// TwinCAT 3 PLC project Development
// ProgramVersion: 3.1.4026.14
// CompilerDefines: release,VISU_USEPROPERTYINFO
// libraries:
//   Tc2_Drive, * (Beckhoff Automation GmbH)
//   Tc2_EtherCAT, * (Beckhoff Automation GmbH)
//   Tc2_MC2, * (Beckhoff Automation GmbH)
//   Tc2_MC2_Drive, * (Beckhoff Automation GmbH)
//   Tc2_Standard, * (Beckhoff Automation GmbH)
//   Tc2_System, * (Beckhoff Automation GmbH)
//   Tc2_Utilities, * (Beckhoff Automation GmbH)
//   Tc3_Element, * (Zerlauth)
//   Tc3_IPCDiag, * (Beckhoff Automation GmbH)
//   Tc3_Module, * (Beckhoff Automation GmbH)
// project tree:
//   GVLs/ IO.TcGVL (not stored)
//   InDevelopment/Axis/ FB_Axis.TcPOU (not stored), F_TcError.TcPOU (not stored), I_Axis.TcIO (not stored)
//   InDevelopment/Contactor/ FB_Contactor.TcPOU
//   InDevelopment/Cylinder/ FB_Cylinder.TcPOU, ST_CylinderOptions.TcDUT (not stored)
//   InDevelopment/ FB_ComponentEX.TcPOU, FB_EthercatDiagnostic.TcPOU (not stored)
//   InDevelopment/PnozMulti/ FB_PnozMulti.TcPOU
//   Modules/ FB_Module01.TcPOU, FB_Machine.TcPOU (not stored), FB_Module02.TcPOU
//   / PlcTask.TcTTO (not stored)
//   POUs/ FB_ComponentT.TcPOU, MAIN.TcPOU
// real-time tasks:
//   TASK PlcTask: cycle T#500ms, priority 21, ADS port 351
//   TASK UnitTestTask: cycle T#1ms, priority 1, ADS port 350
// motion (NC):
//   TASK NC-Task 1 SAF: cycle T#2ms, priority 4, ADS port 501
//   TASK NC-Task 1 SVB: cycle T#10ms, priority 8, ADS port 511
//   AXIS Achse 1 (id 1)
//     OtherSettings: AllowMotionCmdToSlave=true
//     encoder EncType=1
//     drive DrvType=5
//       Analog: TorqueSetpointScale=10, ScaleFactorActTorque=0.1
//       TimeComp: TaskDelayCycles=1
//     controller CtrType=1
//       CtrPara: PriorControlFactor=1
//         Observer: BandWidth=20
// I/O:
//   DEVICE Gerät 1 (EtherCAT) (disabled), AmsNetId 10.58.50.38.2.1
//     Klemme 1 (EK1100) [EK1100 EtherCAT-Koppler (2A E-Bus)]
//     Box 2 (EP1008-0001) [EP1008-0001 8 K. Dig. Eingang 24V, 3ms, M8]
// variable links:
//   Development/Development Instance <-> Device 1 (EtherCAT)
//     PlcTask Inputs/MAIN.fbMachine.fbEthercatDiagnostic.AmsNetID <-> InfoData/AmsNetId

// ---- InDevelopment/Contactor/FB_Contactor.TcPOU
FUNCTION_BLOCK FB_Contactor EXTENDS FB_Element
VAR_INPUT
	bInput				AT%I*: BOOL;
END_VAR
VAR_OUTPUT
	bOutput				AT%I*: BOOL;
END_VAR
VAR
END_VAR

super^();

METHOD PROTECTED M_Running
IF bOutput THEN
	IF bInput  THEN
		;
	ELSE
		P_Event.M_Fatal('Feedback wrong state %s', 0);		
	END_IF
END_IF
END_METHOD

METHOD PROTECTED M_Starting : BOOL (* Return state complete*)
IF bOutput THEN
	IF bInput THEN
		M_Starting:= TRUE;
	ELSE
		P_Event.M_Fatal('Feedback wrong state %s', 0);
	END_IF
ELSE
	IF bInput THEN
		P_Event.M_Fatal('Feedback wrong state %s', 0);
	ELSE
		bOutput:= TRUE;
	END_IF	
	
END_IF
END_METHOD

END_FUNCTION_BLOCK

// ---- InDevelopment/Cylinder/FB_Cylinder.TcPOU
FUNCTION_BLOCK FB_Cylinder EXTENDS FB_Element
VAR_INPUT
	stOptions:				ST_CylinderOptions;
END_VAR
VAR_OUTPUT
END_VAR
VAR
	bInHomePosition			AT%I*:		BOOL;
	bInWorkPosition			AT%I*:		BOOL;
	bToHomePosition			AT%Q*:		BOOL;
	bToWorkPosition			AT%Q*:		BOOL;
	fbHomePositon:			FB_Debounce;
	fbWorkPositon:			FB_Debounce;
	fbStarup:				TON;
	fbTimeout:				TON;
END_VAR

SUPER^();

METHOD PROTECTED M_Aborting : BOOL (* Return*)
bToHomePosition:= FALSE;
bToWorkPosition:= FALSE;
M_Aborting:= TRUE;
END_METHOD

METHOD PROTECTED M_Execute : BOOL // Return state complete
VAR_INPUT
END_VAR
fbHomePositon(bInput:= bInHomePosition);
fbWorkPositon(bInput:= bInWorkPosition);
fbTimeout(PT:= stOptions.tTimeout);
END_METHOD

METHOD PROTECTED M_Starting : BOOL // Return state complete
VAR_INPUT
END_VAR
IF SUPER^.M_Starting() THEN
	fbHomePositon.tTime:= stOptions.tDebounce;
	fbWorkPositon.tTime:= stOptions.tDebounce;
	// Check positons
	IF bToHomePosition AND bToWorkPosition THEN
		IF stOptions.tStartup <> T#0S THEN
			fbStarup(In:= TRUE, PT:= stOptions.tStartup);
			IF fbStarup.Q THEN
				fbStarup(In:= FALSE);
				bToHomePosition:= FALSE;
				bToWorkPosition:= FALSE;
				M_Starting:= TRUE;		
			END_IF
		ELSE
			M_Starting:= TRUE;	
		END_IF
	ELSIF bToHomePosition THEN
		IF NOT bInHomePosition THEN
			P_Event.M_AddSTRING(fbReflection.P_ID);
			P_Event.M_AddSTRING(stOptions.sHomePosition);
			P_Event.M_Error('Cylinder not in Home Positon (%s-%s)', 0);
		ELSIF bInWorkPosition THEN
			P_Event.M_AddSTRING(fbReflection.P_ID);
			P_Event.M_AddSTRING(stOptions.sWorkPosition);
			P_Event.M_Error('Cylinder in Work Positon (%s-%s)', 0);
		ELSE
			M_Starting:= TRUE;	
		END_IF
	ELSIF bToWorkPosition THEN
		IF NOT bInWorkPosition THEN
			P_Event.M_AddSTRING(fbReflection.P_ID);
			P_Event.M_AddSTRING(stOptions.sWorkPosition);
			P_Event.M_Error('Cylinder not in Work Positon (%s-%s)', 0);				
		ELSIF bInHomePosition THEN
			P_Event.M_AddSTRING(fbReflection.P_ID);
			P_Event.M_AddSTRING(stOptions.sHomePosition);
			P_Event.M_Error('Cylinder not in Home Positon (%s-%s)', 0);
		ELSE
			M_Starting:= TRUE;	
		END_IF
	ELSE
		IF bInWorkPosition THEN
			bToWorkPosition:= TRUE;
			M_Starting:= TRUE;
		ELSIF bInHomePosition THEN
			bToHomePosition:= TRUE;
			M_Starting:= TRUE;
		ELSIF stOptions.tStartup <> T#0S THEN		
			bToHomePosition:= TRUE;
			bToWorkPosition:= TRUE;
		ELSE
			M_Starting:= TRUE;
		END_IF
	END_IF
END_IF
END_METHOD

METHOD PUBLIC M_ToHome : BOOL
VAR_INPUT
END_VAR
IF bToWorkPosition THEN
	fbTimeout(IN:= FALSE);
	bToHomePosition:= TRUE;
	bToWorkPosition:= FALSE;

ELSIF bToHomePosition  THEN
	IF NOT fbWorkPositon.P_Value AND fbHomePositon.P_Value THEN
		M_ToHome:= TRUE;
	ELSE
		fbTimeout.IN:= TRUE;
		IF fbTimeout.Q THEN
			IF fbWorkPositon.P_Value THEN
				P_Event.M_AddSTRING(fbReflection.P_ID);
				P_Event.M_AddSTRING(stOptions.sWorkPosition);
				P_Event.M_Error('Cylinder Work Positon not left (%s%s)', 1120);				

			ELSIF NOT fbHomePositon.P_Value THEN
				P_Event.M_AddSTRING(fbReflection.P_ID);
				P_Event.M_AddSTRING(stOptions.sWorkPosition);
				P_Event.M_Error('Cylinder Home Positon not reached (%s%s)', 1121);
	
			END_IF
		END_IF
	END_IF
END_IF
END_METHOD

METHOD PUBLIC M_ToWork : BOOL
VAR_INPUT
END_VAR
IF bToHomePosition THEN
	fbTimeout(IN:= FALSE);
	bToHomePosition:= FALSE;
	bToWorkPosition:= TRUE;	

ELSIF bToWorkPosition  THEN
	IF fbWorkPositon.P_Value AND NOT fbHomePositon.P_Value THEN
		M_ToWork:= TRUE;
	ELSE
		fbTimeout.IN:= TRUE;
		IF fbTimeout.Q THEN
			IF NOT fbWorkPositon.P_Value THEN
				P_Event.M_AddSTRING(fbReflection.P_ID);
				P_Event.M_AddSTRING(stOptions.sWorkPosition);
				P_Event.M_Error('Cylinder Work Positon not reached (%s%s)', 1122);				

			ELSIF fbHomePositon.P_Value THEN
				P_Event.M_AddSTRING(fbReflection.P_ID);
				P_Event.M_AddSTRING(stOptions.sWorkPosition);
				P_Event.M_Error('Cylinder Home Positon not left (%s%s)', 1122);		

			END_IF
		END_IF
	END_IF
END_IF
END_METHOD

{attribute 'suppress_wrn_C0410'}
PROPERTY PUBLIC P_Options : REFERENCE TO ST_CylinderOptions
GET
P_Options ref= stOptions;
END_GET
END_PROPERTY

END_FUNCTION_BLOCK

// ---- InDevelopment/FB_ComponentEX.TcPOU
FUNCTION_BLOCK FB_ComponentEX EXTENDS FB_Element
VAR_INPUT
END_VAR
VAR_OUTPUT
END_VAR
VAR
	bError:			BOOL;
	bAbort:			BOOL;
	bStop:			BOOL;
	bInformation:	BOOL;
	bWarning:		BOOL;
END_VAR

SUPER^();

METHOD PROTECTED M_Execute : BOOL
VAR_INPUT
END_VAR
CASE fbSequence.P_Number OF
	E_Sequence.Start:
		fbSequence.M_Await('Start', 0, T#0S, T#0S, TRUE, TRUE, 10);
	
	10:
		fbSequence.M_Await('Step 10',0,  T#0S, T#0S, TRUE, TRUE, 20);
		
	20:
		fbSequence.M_Await('Step 20',0,  T#0S, T#0S, FALSE, TRUE, E_Sequence.Done);	
		
	E_Sequence.Done:
		fbSequence.M_Reset();
		
END_CASE

IF bAbort THEN
	bAbort:= FALSE;
	fbEvent.M_AddSTRING('1');
	fbEvent.M_AddSTRING('2');
	fbEvent.M_AddSTRING('3');
	fbEvent.M_Fatal('First Error Abort %s %s %s', 6);
END_IF

IF bStop THEN
	bStop:= FALSE;
	fbEvent.M_AddSTRING('a');
	fbEvent.M_AddSTRING('b');
	fbEvent.M_AddSTRING('c');
	fbEvent.M_Error('First Error Stop', 7);
END_IF

IF bInformation THEN
	fbEvent.M_Info('Info', 12);	
END_IF

IF bWarning THEN
	fbEvent.M_Warning('Warning', 13);	
END_IF
END_METHOD

END_FUNCTION_BLOCK

// ---- InDevelopment/PnozMulti/FB_PnozMulti.TcPOU
FUNCTION_BLOCK FB_PnozMulti EXTENDS FB_Element
VAR_INPUT
END_VAR
VAR_OUTPUT
END_VAR
VAR
	bOK:					BOOL:= TRUE;
	bReset:					BOOL;
	fbReset:				TON:= (PT:= T#1S);
END_VAR

SUPER^();

METHOD PROTECTED M_Resetting : BOOL // Return state complete
VAR_INPUT
END_VAR
SUPER^.M_Resetting();
bReset:= TRUE;
fbReset(IN:= TRUE, PT:= T#1S);
IF fbReset.Q THEN
	bReset:= FALSE;
	M_Resetting:= TRUE;
END_IF
END_METHOD

METHOD PROTECTED M_Running
IF NOT bOK THEN
	P_Event.M_AddSTRING(fbReflection.P_ID);
	P_Event.M_Fatal('PnozMulti no ok Signal (%s)', 0);
END_IF
END_METHOD

END_FUNCTION_BLOCK

// ---- Modules/FB_Module01.TcPOU
FUNCTION_BLOCK FB_Module01 EXTENDS FB_Module
VAR_INPUT
END_VAR
VAR_OUTPUT
END_VAR
VAR
END_VAR

// https://peterzerlauth.com/
SUPER^();

METHOD PROTECTED M_Running
VAR_INPUT
END_VAR
END_METHOD

METHOD PROTECTED M_Starting : BOOL
VAR_INPUT
END_VAR
M_Starting:= SUPER^.M_Starting();
END_METHOD

METHOD PROTECTED M_Stopping : BOOL // Return state complete
VAR_INPUT
END_VAR
// State Stopping
M_Stopping:= SUPER^.M_Stopping();
END_METHOD

END_FUNCTION_BLOCK

// ---- Modules/FB_Module02.TcPOU
FUNCTION_BLOCK FB_Module02 EXTENDS FB_Module
VAR_INPUT
END_VAR
VAR_OUTPUT
END_VAR
VAR
	fbPnozMulti:				FB_PnozMulti;
	fbComponent0:				FB_ComponentEx;
	fbComponent1:				FB_ComponentEx;
	fbContactor:				FB_Contactor;
	fbCylinder:					FB_Cylinder;
END_VAR

// https://peterzerlauth.com/
SUPER^();

fbComponent0();
fbComponent1();
fbContactor();
fbCylinder();
fbPnozMulti();

fbContactor.bInput:= fbContactor.bOutput;

METHOD PROTECTED M_Execute : BOOL
VAR_INPUT
END_VAR
VAR
	bReturn:					BOOL:= TRUE;
END_VAR
CASE fbSequence.P_Number OF
	E_Sequence.Start:
		bReturn:= TRUE;
		fbSequence.M_Await('Start 0', 0,  T#0S , T#1S, TRUE, bReturn, 10);
	
	10:
		bReturn:= TRUE;
		fbSequence.M_Await('Step 10', 0,  T#0S, T#0S, TRUE, bReturn, 20);
		
	20:
		bReturn:= TRUE;
		fbSequence.M_Await('Step 20', 0,  T#1S, T#0S, FALSE, bReturn, E_Sequence.Done);
		IF fbSequence.P_Timeout THEN
			fbEvent.M_Error('Overrride timeout error', 0);
		END_IF
		
	E_Sequence.Done:
		fbSequence.M_Reset();

END_CASE
END_METHOD

METHOD PROTECTED M_Idle : BOOL (* Return*)
SUPER^.M_Idle();

fbLevel4.M_Attach(fbPnozMulti);
fbLevel3.M_Attach(fbComponent0);
fbLevel3.M_Attach(fbComponent1);
fbLevel2.M_Attach(fbPnozMulti);
fbLevel2.M_Attach(fbContactor);
fbLevel1.M_Attach(fbCylinder);
END_METHOD

END_FUNCTION_BLOCK

// ---- POUs/FB_ComponentT.TcPOU
FUNCTION_BLOCK FB_ComponentT EXTENDS FB_Element
VAR_INPUT
END_VAR
VAR_OUTPUT
END_VAR
VAR
	bAbort: BOOL;
END_VAR

super^();

METHOD PROTECTED M_Execute : BOOL (* Return*)

IF bAbort THEN
	P_Event.M_Fatal('msg', 0);
END_IF
END_METHOD

END_FUNCTION_BLOCK

// ---- POUs/MAIN.TcPOU
PROGRAM MAIN
VAR
	bTest:				BOOL;
	fbMachine:			FB_Machine;
	fbModule1:			FB_Module01;
	fbModule2:			FB_Module02;
	
	fbComponent1:		FB_ComponentT;
	fbComponent2:		FB_ComponentT;	
	bInit: 				BOOL:= TRUE;
	exceptionCode: 		__SYSTEM.ExceptionCode;
	exception: 			__SYSTEM.ExceptionCode;
	fbFileLogger:		FB_FileLogger<10>:= (sPathName:= 'C:\Temp\log.txt');
	stEvent: 			Tc3_Element.ST_Event;
	bLog: BOOL;
END_VAR

bTest:= NOT bTest;

__TRY
	fbMachine();
	fbModule1();
	fbModule2();


	fbComponent1();
	fbComponent2();
__CATCH(exceptionCode)
 exception:= exceptionCode;
__ENDTRY




IF bInit THEN
	bInit:= False;
	fbComponent1.P_Event.P_Observer.M_Attach(fbComponent2);
	fbComponent2.P_Event.P_Observer.M_Attach(fbComponent1);
END_IF


fbFileLogger();

IF bLog THEN
	bLog:= FALSE;
	stEvent.nID:= 10;
	stEvent.eEventType:= E_Event.Error;
	stEvent.sInstance:= 'Instance';
	stEvent.sClass:= 'Class';
	stEvent.sMessage:= 'Message';
	stEvent.tTimestamp:= DT#2025-01-01-00:00;
	fbFileLogger.M_Log(stEvent);
END_IF

END_PROGRAM
